TYPE st_OutRobotMove :
STRUCT
	Clip				: E_OutRobotClip;
	OutRobotPoint		: E_OutRobotPoint;
	Handshake			: ST_HandshakeBase;
END_STRUCT
END_TYPE

(* stored: Version 1.1.0.1, ProductVersion 3.1.4024.13
   DUT st_OutRobotMove: Id {5acc579e-17da-428c-b6f3-772b12bc4a84} *)
